PROGRAM Grabber_OOR_Timeout
VAR
END_VAR

Timers.GrabberOOR(IN:= Shuttle.Grabber_OOR_Timeout, PT:= T#5S, Q=> , ET=> );

IF Shuttle.ExtensionComplete THEN

	IF Otto.PickupLocation3 AND 
		(Shuttle.GrabberLoadNotInGrabRange[1] OR Shuttle.GrabberLoadNotInGrabRange[2]) THEN 	
		
		Shuttle.Grabber_OOR_Timeout		:= TRUE;
		
	ELSE
		
		Shuttle.Grabber_OOR_Timeout		:= FALSE;
		
	
	END_IF
	
ELSE
	
	Shuttle.Grabber_OOR_Timeout		:= FALSE;

END_IF

IF Timers.GrabberOOR.Q THEN
	
	Shuttle.Grabber_OOR		:= TRUE;

END_IF

END_PROGRAM

(* stored: Version 1.1.0.1, ProductVersion 3.1.4024.9
   POU Grabber_OOR_Timeout: Id {b8f0b067-0d52-4a70-b1fc-b9e3606b9621}, SpecialFunc None *)
